{attribute 'GeneratedUsingTerminal: AMP8000-0030-0103-0103'}
{attribute addProperty BoxType "AMP8000-0030-0103-0103"}
{attribute addProperty Id "DeviceMain_OutputsDeviceMain_Outputs_650F34862"}
{attribute addProperty CRC "1847948663"}
{attribute addProperty Size "2"}
TYPE Device_6E257577 :
STRUCT
	{attribute addProperty Name "DeviceMain_Outputs"}
	DeviceMain_Outputs  : DeviceMain_Outputs_650F3486;
END_STRUCT
END_TYPE

(* stored: Version 1.2.0.0, ProductVersion 3.1.4024.9
   DUT Device_6E257577: Id {d2f27fa7-ac1a-40ae-a6c0-c0f5973d28b1} *)
